Fanuc KAREL source: wuserelaccel.kl

PROGRAM wuserelaccel
%NOLOCKGROUP
VAR
  p : POSITION
  q : POSITION
  i : INTEGER
  r : REAL
BEGIN
  WITH $USERELACCEL = TRUE MOVE TO p
END wuserelaccel
